// TIA Portal V17 export
// export: Created 2026-04-13T11:12:45.155941Z, ExportSetting WithDefaults, DisplayName Totally Integrated Automation Portal, DisplayVersion V17 Update 4, DisplayName TIA Portal Openness, DisplayVersion V17 Update 4, DisplayName TIA Portal Version Control Interface, DisplayVersion V17, DisplayName SINAMICS Startdrive Advanced, DisplayVersion V17, DisplayName SINAMICS Startdrive G130, G150, S120, S150, SINAMICS MV, S210, DisplayVersion V17, DisplayName SINAMICS Startdrive G110M, G120, G120C, G120D, G120P, G115D, DisplayVersion V17, DisplayName STEP 7 Professional, DisplayVersion V17 Update 4, DisplayName STEP 7 Safety, DisplayVersion V17, DisplayName WinCC Professional, DisplayVersion V17 Update 4
VAR_GLOBAL   // PLC tag table "Alarm"
   A备用报警1 AT %M23.6 : Bool;
   AWK温控高温报警 AT %M37.7 : Bool;
   AKY空压低压信号 AT %M31.3 : Bool;
   ASS输送加热报警 AT %M34.7 : Bool;
   AWH雾化关报警 AT %M37.0 : Bool;
   AWH雾化开报警 AT %M37.1 : Bool;
   ABD布袋压差高报 AT %M20.2 : Bool;
   ABD布袋压差高高报 AT %M20.3 : Bool;
   AJF进风压差高高报 AT %M28.7 : Bool;
   AJF进风压差高报 AT %M28.6 : Bool;
   ATN塔内压力低报 AT %M36.4 : Bool;
   ATN塔内压力高报 AT %M36.6 : Bool;
   AJF进风温度高报 AT %M29.4 : Bool;
   AJF进风温度故障 AT %M29.3 : Bool;
   ACF出风温度高报 AT %M22.3 : Bool;
   ACF出风温度故障 AT %M22.1 : Bool;
   AWH雾化进氮低报 AT %M37.5 : Bool;
   AWQ尾气温度高报 AT %M38.1 : Bool;
   报警1 AT %MW20 : Word;
   ALD冷冻水关报警 AT %M31.4 : Bool;
   ACF出风温度过低 AT %M22.2 : Bool;
   AYH氧含量运行故障 AT %M39.2 : Bool;
   AJT急停报警 AT %M30.5 : Bool;
   报警2 AT %MW22 : Word;
   AJD进氮压力低报 AT %M27.3 : Bool;
   ATN塔内压力高高报 AT %M36.7 : Bool;
   AJF进风温度高高报 AT %M29.5 : Bool;
   ACF出风温度高高报 AT %M22.4 : Bool;
   ATN塔内压力低低报 AT %M36.3 : Bool;
   AWQ尾气温度高高报 AT %M38.2 : Bool;
   AGD管道压力高报 AT %M26.1 : Bool;
   AGD管道压力高高报 AT %M26.2 : Bool;
   AWQ尾气故障 AT %M38.0 : Bool;
   ALX离心雾化故障 AT %M31.7 : Bool;
   AJX机械温控故障 AT %M30.6 : Bool;
   AQT气体检测低报 AT %M32.4 : Bool;
   AQT气体检测低低报 AT %M32.3 : Bool;
   AWK温控未通信 AT %M37.6 : Bool;
   AHS回收罐1报警 AT %M26.7 : Bool;
   AHS回收罐2报警 AT %M27.0 : Bool;
   AJL进料泵故障报警 AT %M30.1 : Bool;
   AYF引风机报警 AT %M38.5 : Bool;
   AJB搅拌电机报警 AT %M27.1 : Bool;
   AQL气流雾化阀开报警 AT %M32.2 : Bool;
   AQL气流雾化阀关报警 AT %M32.1 : Bool;
   AYJ一级出料上阀开报警 AT %M39.6 : Bool;
   AYJ一级出料上阀关报警 AT %M39.5 : Bool;
   AYJ一级出料下阀开报警 AT %M40.0 : Bool;
   AYJ一级出料下阀关报警 AT %M39.7 : Bool;
   AEJ二级出料上阀开报警 AT %M24.2 : Bool;
   AEJ二级出料上阀关报警 AT %M24.1 : Bool;
   AEJ二级出料下阀开报警 AT %M24.4 : Bool;
   AEJ二级出料下阀关报警 AT %M24.3 : Bool;
   ACC除尘出料上阀开报警 AT %M21.5 : Bool;
   ACC除尘出料上阀关报警 AT %M21.4 : Bool;
   ACC除尘出料下阀开报警 AT %M21.7 : Bool;
   ACC除尘出料下阀关报警 AT %M21.6 : Bool;
   AKS开式排风隔断阀开报警 AT %M31.0 : Bool;
   AKS开式排风隔断阀关报警 AT %M30.7 : Bool;
   ABS闭式排风隔断阀开报警 AT %M21.1 : Bool;
   ABS闭式排风隔断阀关报警 AT %M21.0 : Bool;
   AKS开式进风隔断阀开报警 AT %M31.2 : Bool;
   AKS开式进风隔断阀关报警 AT %M31.1 : Bool;
   ABS闭式进风隔断阀开报警 AT %M21.3 : Bool;
   ABS闭式进风隔断阀关报警 AT %M21.2 : Bool;
   AYJ一级冷却水阀开报警 AT %M39.4 : Bool;
   AYJ一级冷却水阀关报警 AT %M39.3 : Bool;
   AEJ二级冷冻水阀开报警 AT %M24.0 : Bool;
   AEJ二级冷冻水阀关报警 AT %M23.7 : Bool;
   AYJ一级排液阀开报警 AT %M40.2 : Bool;
   AYJ一级排液阀关报警 AT %M40.1 : Bool;
   AEJ二级排液阀开报警 AT %M24.6 : Bool;
   AEJ二级排液阀关报警 AT %M24.5 : Bool;
   ACW除雾排液阀开报警 AT %M23.1 : Bool;
   ACW除雾排液阀关报警 AT %M23.0 : Bool;
   ARJ溶剂回收排放阀开报警 AT %M33.3 : Bool;
   ARJ溶剂回收排放阀关报警 AT %M33.2 : Bool;
   AXY泄压阀开报警 AT %M38.4 : Bool;
   AXY泄压阀关报警 AT %M38.3 : Bool;
   AJF进风冷却水阀开报警 AT %M28.2 : Bool;
   AJF进风冷却水阀关报警 AT %M28.1 : Bool;
   ASS输送进风阀开报警 AT %M35.4 : Bool;
   ASS输送进风阀关报警 AT %M35.3 : Bool;
   ASS输送出料上阀开报警 AT %M34.4 : Bool;
   ASS输送出料上阀关报警 AT %M34.3 : Bool;
   ASS输送出料下阀开报警 AT %M34.6 : Bool;
   ASS输送出料下阀关报警 AT %M34.5 : Bool;
   ATD塔顶清洗球阀开报警 AT %M36.2 : Bool;
   ATD塔顶清洗球阀关报警 AT %M36.1 : Bool;
   AQX清洗伸缩气缸开报警 AT %M32.6 : Bool;
   AQX清洗伸缩气缸关报警 AT %M32.5 : Bool;
   ABD补氮阀开报警 AT %M20.5 : Bool;
   ABD补氮阀关报警 AT %M20.4 : Bool;
   AJD进氮阀开报警 AT %M27.6 : Bool;
   AJD进氮阀关报警 AT %M27.5 : Bool;
   ASF送风机报警 AT %M33.7 : Bool;
   AJF进风保护温度报警 AT %M27.7 : Bool;
   ASS输送保护温度报警 AT %M34.2 : Bool;
   ABP爆破片1反馈报警 AT %M20.6 : Bool;
   ABP爆破片2反馈报警 AT %M20.7 : Bool;
   ASN室内排水开反馈报警 AT %M34.1 : Bool;
   ASN室内排水关反馈报警 AT %M34.0 : Bool;
   ADJ电加热报警 AT %M23.5 : Bool;
   AWH雾化油压低报 AT %M37.3 : Bool;
   AWH雾化油压低低报 AT %M37.2 : Bool;
   AJD进氮压力低低报 AT %M27.2 : Bool;
   AFD阀导气压低报 AT %M25.3 : Bool;
   AFD阀导气压低低报 AT %M25.2 : Bool;
   AJF进风压差低报 AT %M28.4 : Bool;
   ACF出风高效高报 AT %M22.6 : Bool;
   ACF出风高效高高报 AT %M22.7 : Bool;
   ACF出风高效低报 AT %M22.5 : Bool;
   ASS输送高效高报 AT %M35.7 : Bool;
   ASS输送高效高高报 AT %M36.0 : Bool;
   ASF输送高效低报 AT %M33.6 : Bool;
   AHF回风温度高报 AT %M26.5 : Bool;
   AHF回风温度高高报 AT %M26.6 : Bool;
   AJF进风冷却水流量低报警 AT %M28.0 : Bool;
   ALD冷冻水流量低报警 AT %M31.5 : Bool;
   ALQ冷却水流量低报警 AT %M31.6 : Bool;
   ABD布袋压差低报 AT %M20.0 : Bool;
   AJF进风流量计故障 AT %M29.2 : Bool;
   AJL进料流量故障 AT %M30.4 : Bool;
   AJF进风压差变送器故障 AT %M28.5 : Bool;
   ACF出风压差变送器故障 AT %M22.0 : Bool;
   ABD布袋压差变送器故障 AT %M20.1 : Bool;
   ASS输送高效压差变送器故障 AT %M35.6 : Bool;
   AJL进料压力故障 AT %M29.6 : Bool;
   ATN塔内压力故障 AT %M36.5 : Bool;
   AGD管道压力变送器故障 AT %M26.0 : Bool;
   AJD进氮压力故障 AT %M27.4 : Bool;
   AFK放空比例反馈故障 AT %M25.7 : Bool;
   AJF进风加热比例反馈故障 AT %M28.3 : Bool;
   AHF回风加热比例反馈故障 AT %M26.3 : Bool;
   AWH雾化油压故障 AT %M37.4 : Bool;
   AYH氧含仪1故障 AT %M38.6 : Bool;
   AYH氧含仪2故障 AT %M38.7 : Bool;
   AYJ一级溶剂液位计故障 AT %M40.5 : Bool;
   AEJ二级溶剂液位计故障 AT %M25.1 : Bool;
   ACW除雾溶剂液位计故障 AT %M23.4 : Bool;
   AFD阀岛气压故障报警 AT %M25.6 : Bool;
   AJL进料压力高报 AT %M29.7 : Bool;
   AJL进料压力高高报 AT %M30.0 : Bool;
   ASS输送温度高高报 AT %M35.2 : Bool;
   ASS输送温度高报 AT %M35.1 : Bool;
   ASS输送温度故障报警 AT %M35.0 : Bool;
   AHF回风温度故障报警 AT %M26.4 : Bool;
   ASS输送高效低报 AT %M35.5 : Bool;
   AYJ一级液位计高报 AT %M40.3 : Bool;
   AYJ一级液位计高高报 AT %M40.4 : Bool;
   AEJ二级液位计高报 AT %M24.7 : Bool;
   AEJ二级液位计高高报 AT %M25.0 : Bool;
   ACW除雾液位计高报 AT %M23.2 : Bool;
   ACW除雾液位计高高报 AT %M23.3 : Bool;
   AFD阀岛气压低报 AT %M25.5 : Bool;
   AFD阀岛气压低低报 AT %M25.4 : Bool;
   APY排液流量低报警 AT %M32.0 : Bool;
   ASF输送风机故障报警 AT %M33.5 : Bool;
   ASF输送加热故障报警 AT %M33.4 : Bool;
   AYH氧含仪高报 AT %M39.0 : Bool;
   AYH氧含仪高高报 AT %M39.1 : Bool;
   AJF进风流量低低报 AT %M29.0 : Bool;
   AJF进风流量低报 AT %M29.1 : Bool;
   AQZ前置液位低报 AT %M33.0 : Bool;
   AQZ前置液位低低报 AT %M32.7 : Bool;
   AQZ前置液位计故障 AT %M33.1 : Bool;
   AJL进料流量低报 AT %M30.3 : Bool;
   AJL进料流量低低报 AT %M30.2 : Bool;
   报警3 AT %MW24 : Word;
   报警4 AT %MW26 : Word;
   报警5 AT %MW28 : Word;
   报警6 AT %MW30 : Word;
   报警7 AT %MW32 : Word;
   报警8 AT %MW34 : Word;
   报警9 AT %MW36 : Word;
   报警10 AT %MW38 : Word;
   报警11 AT %MW40 : Word;
   报警12 AT %MW42 : Word;
   AKS开式自动自检不通过 AT %M40.6 : Bool;
   ACIP缺水报警 AT %M40.7 : Bool;
   ARJ溶剂排液泵开报警 AT %M41.0 : Bool;
   ARJ溶剂排液泵关报警 AT %M41.1 : Bool;
END_VAR
